// TIA Portal V20 export
DATA_BLOCK "BK18"   // DB312
// stored: MemoryReserve 100
   VAR
      "X10-1.ANODE MANDREL REAR Y AXIS LIMIT SENSOR(-)" : Bool := TRUE;
      "X11-1.ANODE MANDREL REAR Y AXIS LIMIT SENSOR(+)" : Bool := TRUE;
      "X12-1.ANODE MANDREL REAR Z AXIS LIMIT SENSOR(-)" : Bool := TRUE;
      "X13-1.ANODE MANDREL REAR Z AXIS LIMIT SENSOR(+)" : Bool := TRUE;
      "X14-1.ANODE MANDREL FRONT Y AXIS LIMIT SENSOR(-)" : Bool := TRUE;
      "X15-1.ANODE MANDREL FRONT Y AXIS LIMIT SENSOR(+)" : Bool := TRUE;
      "X16-1.ANODE MANDREL FRONT Z AXIS LIMIT SENSOR(-)" : Bool := TRUE;
      "X17-1.ANODE MANDREL FRONT Z AXIS LIMIT SENSOR(+)" : Bool := TRUE;
      "X10-2.ANODE MANDREL REAR Y AXIS HOME SENSOR" : Bool := TRUE;
      "X11-2.SPARE" : Bool := FALSE;
      "X12-2.ANODE MANDREL REAR Z AXIS HOME SENSOR" : Bool := TRUE;
      "X13-2.SPARE" : Bool := FALSE;
      "X14-2.ANODE MANDREL FRONT Y AXIS HOME SENSOR" : Bool := TRUE;
      "X15-2.SPARE" : Bool := FALSE;
      "X16-2.ANODE MANDREL FRONT Z AXIS HOME SENSOR" : Bool := TRUE;
      "X17-2.SPARE" : Bool := FALSE;
   END_VAR
BEGIN
END_DATA_BLOCK
